// TIA Portal V18 export
// export: Created 2026-06-08T03:54:35.0001352Z, ExportSetting WithDefaults, DisplayName Totally Integrated Automation Portal, DisplayVersion V18, DisplayName TIA Portal Openness, DisplayVersion V18, DisplayName TIA Portal Version Control Interface, DisplayVersion V18, DisplayName STEP 7 Professional, DisplayVersion V18, DisplayName STEP 7 Safety, DisplayVersion V18, DisplayName WinCC Professional, DisplayVersion V18
FUNCTION "FC_Init_Default_Recipe_PLC2" : Void   // FC51, LAD
{ S7_Optimized_Access := 'TRUE' }
VERSION : 0.1
// stored: AutoNumber true, IsIECCheckEnabled false, SetENOAutomatically false, UDAEnableTagReadback false
BEGIN

REGION Network 1: Kích hoạt nạp recipe mặc định lần đầu scan PLC2
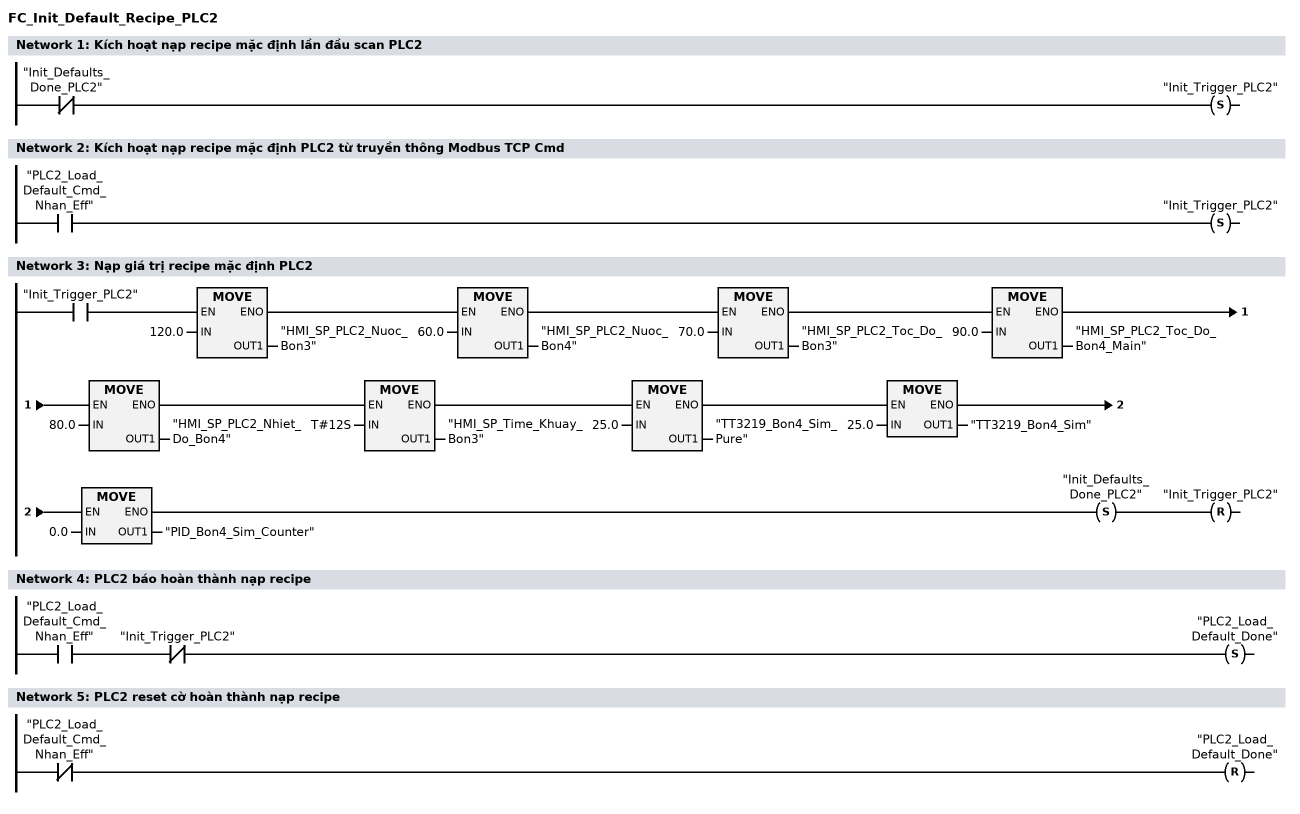
   RUNG wire#powerrail
      I_Contact( "Init_Defaults_Done_PLC2" )
      S_Coil( "Init_Trigger_PLC2" )
   END_RUNG
   // the same network as SCL:
   IF NOT "Init_Defaults_Done_PLC2" THEN "Init_Trigger_PLC2" := TRUE; END_IF;
END_REGION

REGION Network 2: Kích hoạt nạp recipe mặc định PLC2 từ truyền thông Modbus TCP Cmd
   RUNG wire#powerrail
      Contact( "PLC2_Load_Default_Cmd_Nhan_Eff" )
      S_Coil( "Init_Trigger_PLC2" )
   END_RUNG
   // the same network as SCL:
   IF "PLC2_Load_Default_Cmd_Nhan_Eff" THEN "Init_Trigger_PLC2" := TRUE; END_IF;
END_REGION

REGION Network 3: Nạp giá trị recipe mặc định PLC2
   RUNG wire#powerrail
      Contact( "Init_Trigger_PLC2" )
      { S7_GenerateENO := "TRUE" } Move(in := 120.0, out1 => "HMI_SP_PLC2_Nuoc_Bon3")
      { S7_GenerateENO := "TRUE" } Move(in := 60.0, out1 => "HMI_SP_PLC2_Nuoc_Bon4")
      { S7_GenerateENO := "TRUE" } Move(in := 70.0, out1 => "HMI_SP_PLC2_Toc_Do_Bon3")
      { S7_GenerateENO := "TRUE" } Move(in := 90.0, out1 => "HMI_SP_PLC2_Toc_Do_Bon4_Main")
      { S7_GenerateENO := "TRUE" } Move(in := 80.0, out1 => "HMI_SP_PLC2_Nhiet_Do_Bon4")
      { S7_GenerateENO := "TRUE" } Move(in := T#12S, out1 => "HMI_SP_Time_Khuay_Bon3")
      { S7_GenerateENO := "TRUE" } Move(in := 25.0, out1 => "TT3219_Bon4_Sim_Pure")
      { S7_GenerateENO := "TRUE" } Move(in := 25.0, out1 => "TT3219_Bon4_Sim")
      { S7_GenerateENO := "TRUE" } Move(in := 0.0, out1 => "PID_Bon4_Sim_Counter")
      S_Coil( "Init_Defaults_Done_PLC2" )
      R_Coil( "Init_Trigger_PLC2" )
   END_RUNG
   // the same network as SCL:
   // ENO of a box is taken as its EN; it also drops when the box reports an error
   IF "Init_Trigger_PLC2" THEN
       "HMI_SP_PLC2_Nuoc_Bon3" := 120.0;
       "HMI_SP_PLC2_Nuoc_Bon4" := 60.0;
       "HMI_SP_PLC2_Toc_Do_Bon3" := 70.0;
       "HMI_SP_PLC2_Toc_Do_Bon4_Main" := 90.0;
       "HMI_SP_PLC2_Nhiet_Do_Bon4" := 80.0;
       "HMI_SP_Time_Khuay_Bon3" := T#12S;
       "TT3219_Bon4_Sim_Pure" := 25.0;
       "TT3219_Bon4_Sim" := 25.0;
       "PID_Bon4_Sim_Counter" := 0.0;
       "Init_Defaults_Done_PLC2" := TRUE;
       "Init_Trigger_PLC2" := FALSE;
   END_IF;
END_REGION

REGION Network 4: PLC2 báo hoàn thành nạp recipe
   RUNG wire#powerrail
      Contact( "PLC2_Load_Default_Cmd_Nhan_Eff" )
      I_Contact( "Init_Trigger_PLC2" )
      S_Coil( "PLC2_Load_Default_Done" )
   END_RUNG
   // the same network as SCL:
   IF "PLC2_Load_Default_Cmd_Nhan_Eff" AND NOT "Init_Trigger_PLC2" THEN
       "PLC2_Load_Default_Done" := TRUE;
   END_IF;
END_REGION

REGION Network 5: PLC2 reset cờ hoàn thành nạp recipe
   RUNG wire#powerrail
      I_Contact( "PLC2_Load_Default_Cmd_Nhan_Eff" )
      R_Coil( "PLC2_Load_Default_Done" )
   END_RUNG
   // the same network as SCL:
   IF NOT "PLC2_Load_Default_Cmd_Nhan_Eff" THEN "PLC2_Load_Default_Done" := FALSE; END_IF;
END_REGION
END_FUNCTION
